{attribute 'GeneratedUsingTerminal: EL5122-0000-0016'}
{attribute addProperty BoxType "EL5122-0000-0016"}
{attribute addProperty Id "Enable_latch_extern_on_positive_edgeBOOL1Set_counterBOOL1Enable_latch_extern_on_negative_edgeBOOL1Set_software_gateBOOL1Set_counter_on_latch_extern_on_positive_edgeBOOL1Set_counter_on_latch_extern_on_negative_edgeBOOL1"}
{attribute addProperty CRC "2740673020"}
{attribute addProperty Size "6"}
TYPE Control_A35B59FC :
STRUCT
	{attribute addProperty Name "Enable_latch_extern_on_positive_edge"}
	Enable_latch_extern_on_positive_edge : BOOL;
	{attribute addProperty Name "Set_counter"}
	Set_counter : BOOL;
	{attribute addProperty Name "Enable_latch_extern_on_negative_edge"}
	Enable_latch_extern_on_negative_edge : BOOL;
	{attribute addProperty Name "Set_software_gate"}
	Set_software_gate : BOOL;
	{attribute addProperty Name "Set_counter_on_latch_extern_on_positive_edge"}
	Set_counter_on_latch_extern_on_positive_edge : BOOL;
	{attribute addProperty Name "Set_counter_on_latch_extern_on_negative_edge"}
	Set_counter_on_latch_extern_on_negative_edge : BOOL;
END_STRUCT
END_TYPE

(* stored: Version 1.2.0.0, ProductVersion 3.1.4024.9
   DUT Control_A35B59FC: Id {b7d7d0ac-9305-4740-9487-c62fb27e88a5} *)
